// TwinCAT 3 PLC project Untitled1
// ProgramVersion: 3.1.4023.0
// libraries:
//   Tc2_Standard, * (Beckhoff Automation GmbH)
//   Tc2_System, * (Beckhoff Automation GmbH)
//   Tc3_Module, * (Beckhoff Automation GmbH)
// project tree:
//   / PlcTask.TcTTO
//   POUs/ MAIN.TcPOU, POU.TcPOU
// real-time tasks:
//   TASK PlcTask: cycle T#5ms, priority 20, ADS port 350

CONFIGURATION Untitled1
    RESOURCE PLC ON TwinCAT3
        TASK PlcTask(INTERVAL := T#5ms, PRIORITY := 20);
        PROGRAM MAIN WITH PlcTask : MAIN;
    END_RESOURCE
END_CONFIGURATION

// ---- POUs/MAIN.TcPOU
PROGRAM MAIN
VAR
	i: INT;
END_VAR

i:=i+1;

END_PROGRAM

// ---- POUs/POU.TcPOU
FUNCTION_BLOCK POU IMPLEMENTS ITcTask
VAR_INPUT
END_VAR
VAR_OUTPUT
END_VAR
VAR
END_VAR

???(pCnt := ???.Q); // GetCycleCounter
???(IN := ???.GetCycleCounter); // TON

{attribute 'TcTypeSystem'}
{attribute 'no-analysis'}
{attribute 'c++_compatible'}
{attribute 'minimal_input_size' := '4'}
{attribute 'pack_mode' := '4'}
{warning 'add method implementation '}
METHOD GetCurrentDcTime : HRESULT
VAR_INPUT
	pDcTime	: POINTER TO UDINT;
END_VAR
END_METHOD

{attribute 'TcTypeSystem'}
{attribute 'no-analysis'}
{attribute 'c++_compatible'}
{attribute 'minimal_input_size' := '4'}
{attribute 'pack_mode' := '4'}
{warning 'add method implementation '}
METHOD GetCurrentSysTime : HRESULT
VAR_INPUT
	pSysTime	: POINTER TO ULINT;
END_VAR
END_METHOD

{attribute 'TcTypeSystem'}
{attribute 'no-analysis'}
{attribute 'c++_compatible'}
{attribute 'minimal_input_size' := '4'}
{attribute 'pack_mode' := '4'}
{warning 'add method implementation '}
METHOD GetCycleCounter : HRESULT
VAR_INPUT
	pCnt	: POINTER TO ULINT;
END_VAR
END_METHOD

{attribute 'TcTypeSystem'}
{attribute 'no-analysis'}
{attribute 'c++_compatible'}
{attribute 'minimal_input_size' := '4'}
{attribute 'pack_mode' := '4'}
{warning 'add method implementation '}
METHOD GetCycleTime : HRESULT
VAR_INPUT
	pCycleTimeNS	: POINTER TO UDINT;
END_VAR
END_METHOD

{attribute 'TcTypeSystem'}
{attribute 'no-analysis'}
{attribute 'c++_compatible'}
{attribute 'minimal_input_size' := '4'}
{attribute 'pack_mode' := '4'}
{warning 'add method implementation '}
METHOD GetPriority : HRESULT
VAR_INPUT
	pPriority	: POINTER TO UDINT;
END_VAR
END_METHOD

{attribute 'TcTypeSystem'}
{attribute 'no-analysis'}
{attribute 'c++_compatible'}
{attribute 'minimal_input_size' := '4'}
{attribute 'pack_mode' := '4'}
{warning 'add method implementation '}
METHOD TcAddRef : UDINT
END_METHOD

{attribute 'TcTypeSystem'}
{attribute 'no-analysis'}
{attribute 'c++_compatible'}
{attribute 'minimal_input_size' := '4'}
{attribute 'pack_mode' := '4'}
{warning 'add method implementation '}
METHOD TcQueryInterface : HRESULT
VAR_INPUT
	iid	: REFERENCE TO IID;
	pipItf	: POINTER TO PVOID;
END_VAR
END_METHOD

{attribute 'TcTypeSystem'}
{attribute 'no-analysis'}
{attribute 'c++_compatible'}
{attribute 'minimal_input_size' := '4'}
{attribute 'pack_mode' := '4'}
{warning 'add method implementation '}
METHOD TcRelease : UDINT
END_METHOD

END_FUNCTION_BLOCK
